FUNCTION_BLOCK FB_HnltCnLinkage
VAR_INPUT
	stAmbientState : ST_AmbientState;
	
	//control struct for hnlt cn linkage
	controlAutomatic : ST_HnltCnLinkageControl;
END_VAR
VAR_OUTPUT
END_VAR
VAR
	//systems
	HeatPumpSystem : FB_HeatPumpSystem;
	InnerCapillaryTubeMats : FB_InnerCapillaryTubeMats;
	
	//internal variables
	bAlgorithmPermission : BOOL;
END_VAR

//check for algorithm permission
bAlgorithmPermission := controlAutomatic.bAlgorithmPermission_CN AND controlAutomatic.bAlgorithmPermission_HNLT;

//NOTE: heat pump systems contains only two-point actors -> fSetPointAutomatic = 0	
HeatPumpSystem(bSetStatusOnAutomatic := controlAutomatic.bSetStatusOn_HeatPump,
	bAlgorithmPermission := bAlgorithmPermission,
	fSetPointAutomatic := 0);

//NOTE: inner capillary tube mats are always on and recieve desired hall temperature as setpoint
InnerCapillaryTubeMats(bSetStatusOnAutomatic := TRUE,
	bAlgorithmPermission := bAlgorithmPermission,
	fSetPointAutomatic := controlAutomatic.fTargetTemperature_ProductionHall,
	bHeatingModeAutomatic := controlAutomatic.bHeatingMode,
	stAmbientState := stAmbientState);

END_FUNCTION_BLOCK

(* stored: Version 1.1.0.1, ProductVersion 3.1.4024.10
   POU FB_HnltCnLinkage: Id {49b9fb4a-ee7f-4dd8-8511-b340abe8c57d}, SpecialFunc None *)
